FUNCTION Convert_TOD_TO_LINT : BOOL
VAR_INPUT
	in : TOD;
	out : REFERENCE TO LINT;
END_VAR
VAR
	converted : LINT;
END_VAR

converted := TOD_TO_LINT(in);

IF (LINT_TO_TOD(converted) <> in) THEN
	RETURN;
END_IF

out := converted;
Convert_TOD_TO_LINT := TRUE;

END_FUNCTION

(* stored: Version 1.1.0.1, ProductVersion 3.1.4024.12
   POU Convert_TOD_TO_LINT: Id {a74d1bbc-090a-42f9-a50d-a5b9ee83ed12}, SpecialFunc None *)
